// TIA Portal V17 export
// export: Created 2024-09-03T21:54:48.5238419Z, ExportSetting WithDefaults, DisplayName Totally Integrated Automation Portal, DisplayVersion V17 Update 7, DisplayName TIA Portal Openness, DisplayVersion V17 Update 7, DisplayName TIA Portal Version Control Interface, DisplayVersion V17, DisplayName SINAMICS Startdrive Advanced, DisplayVersion V17 SP2, DisplayName SINAMICS Startdrive G110M, G120, G120C, G120D, G120P, G115D, DisplayVersion V17 SP2, DisplayName SINAMICS Startdrive G130, G150, S120, S150, SINAMICS MV, S210, DisplayVersion V17 SP2, DisplayName STEP 7 Professional, DisplayVersion V17 Update 7, DisplayName STEP 7 Safety, DisplayVersion V17 Update 6, DisplayName WinCC Advanced / Unified PC, DisplayVersion V17 Update 7
DATA_BLOCK "CylindersHMI"   // DB50
{ S7_Optimized_Access := 'TRUE' }
VERSION : 0.1
// stored: AutoNumber true, DBAccessibleFromOPCUA true, DBAccessibleFromWebserver true, IsOnlyStoredInLoadMemory false, IsRetainMemResEnabled false, IsWriteProtectedInAS false, MemoryReserve 100
   VAR
      Status : Array[0.."NumberOfCylinders"] of Int;
      SelectedCylinderCylinderCommand : Int := 0;
      SelectedCylinder : Int := 0;
      SelectedCylinderStatus : Int := 0;
      SelectedCylinder_1 : Int := 0;
      SelectedCylinder_2 : Int := 0;
      SelectedCylinder_3 : Int := 0;
      SelectedCylinder_4 : Int := 0;
      SelectedCylinderStatus_1 : Int := 0;
      SelectedCylinderStatus_2 : Int := 0;
      SelectedCylinderStatus_3 : Int := 0;
      SelectedCylinderStatus_4 : Int := 0;
      DisableHMIControl : Bool := FALSE;
      CylinderInfoHMI : Int := -1;
      CylinderInfoHMIAction : Int := 0;
   END_VAR
BEGIN
   Status[0..4] := 257;
   Status[5..6] := 1;
   Status[7..8] := 257;
   Status[9..10] := 1;
   Status[11..14] := 257;
   Status[15..16] := 1;
   Status[17] := 2;
   Status[18] := 1;
   Status[19] := 0;
END_DATA_BLOCK
